FUNCTION_BLOCK QUARTER_TO_E (* quad-state to 4 Events *)
  (* Standard: 61499-2; Description: Copyright (c) 2024 franz This program and the accompanying materials are made available under the terms of the Eclipse Public License 2.0 which is available at https://www.eclipse.org/legal/epl-2.0/ SPDX-License-Identifier: EPL-2.0 *)
  (* Version 1.0, 2024-02-23, franz *)
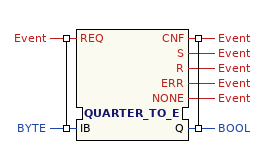
  EVENT_INPUT
    REQ WITH IB; (* Normal Execution Request *)
  END_EVENT
  EVENT_OUTPUT
    CNF WITH Q; (* Execution Confirmation *)
    S; (* Enabled (on, active, etc.) *)
    R; (* Disabled (off, passive, etc.) *)
    ERR; (* Error indicator *)
    NONE; (* Not available or not installed *)
  END_EVENT
  VAR_INPUT
    IB : BYTE := COMMAND_DISABLE; (* 2bit (quarter Byte) Output with 4 States *)
  END_VAR
  VAR_OUTPUT
    Q : BOOL; (* BOOL Output *)
  END_VAR
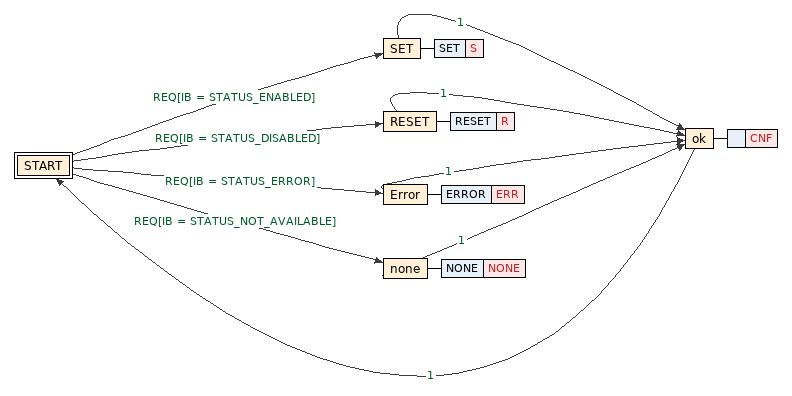
  EC_STATES
    START; (* Initial State *)
    SET : SET -> S;
    RESET : RESET -> R;
    Error : ERROR -> ERR;
    none : NONE -> NONE;
    ok : -> CNF;
  END_STATES
  EC_TRANSITIONS
    START TO SET := REQ[IB = STATUS_ENABLED];
    START TO RESET := REQ[IB = STATUS_DISABLED];
    START TO Error := REQ[IB = STATUS_ERROR];
    START TO none := REQ[IB = STATUS_NOT_AVAILABLE];
    SET TO ok := 1;
    RESET TO ok := 1;
    Error TO ok := 1;
    none TO ok := 1;
    ok TO START := 1;
  END_TRANSITIONS
  ALGORITHM SET IN ST:
Q := TRUE;
  END_ALGORITHM
  ALGORITHM RESET IN ST:
Q := FALSE;
  END_ALGORITHM
  ALGORITHM ERROR IN ST:
Q := FALSE;
  END_ALGORITHM
  ALGORITHM NONE IN ST:
// Q Don't care/take no action (leave function as is)
  END_ALGORITHM
END_FUNCTION_BLOCK
